Universal Robots URScript: LEscript_grind.script

# File: LEscript_grind.script
# Project: LEonard
# Author: Ned Lecky, Lecky Engineering LLC
# Purpose: LEonard Grinding Support

global version_grind = "LEscript_grind.script 2022-11-23"

global grind_ready = True
# grind_contact_enable:  0=No Contact   1=Touch but no tool/coolant on or force  2=Touch, Tool, Coolant, and Force
global grind_contact_enable = 0
global grind_touch_retract_mm = 3       # How far to retract after touch  (we do 2X this for ghrind_contact_enable=1)
global grind_touch_speed_mmps = 0.1     # How fast to go in for the touch
global grind_force_dwell_ms = 500       # How long to dwell after turning force more on
global grind_max_blend_radius_m = 0.010 # Max blend radius to use while grinding
global grind_trial_speed_mmps = 20      # Grinding speed when not really grinding!
global grind_point_frequency_hz = 4     # Points per second to generate in grind_movel

# Current speeds in use for grinding... the angular are computed off the linear
# And the two are blended by draw_to for cylinders
global grind_linear_vel_mps = 0
global grind_linear_accel_mpss = 0
global grind_linear_blend_radius_m = 0
global grind_angular_vel_rps = 0
global grind_angular_accel_rpss = 0
global grind_angular_blend_radius_rad = 0

# Grinding speeds when not in contact
global grind_jog_speed_mmps = 40     # Speed used internally when adjusting and moving around part
global grind_jog_accel_mmpss = 100   # Accel used internally when adjusting and moving around part

# Force mode parameters
global grind_force_mode_damping = 0.0
global grind_force_mode_gain_scaling = 1.0

# Planning points
global p_operator_init = p[0, 0, 0, 0, 0, 0]    # Where we were when operator issued first grind command
global p_contact_init = p[0, 0, 0, 0, 0, 0]     # Where we first contacted the part
global p_contact_center = p[0, 0, 0, 0, 0, 0]   # Computed where center of pattern would be in contact with part

# Set grind variables chosen by command[2]
# Value after set is always returned to socket
def set_grind_variable():
  global grind_ready = False
  socket_send_bool("grind_ready", grind_ready)

  if command[2] == 1:
    global response = "set grind_contact_enable"
    if command[3] >= 0 and command[3] <= 2:
      global grind_contact_enable = ceil(command[3])
    end
    socket_send_number("grind_contact_enable", grind_contact_enable)
  elif command[2] == 2:
    global response = "set grind_touch_retract_mm"
    if command[3] >= 0:
      global grind_touch_retract_mm = ceil(command[3])
    end
    socket_send_number("grind_touch_retract_mm", grind_touch_retract_mm)
  elif command[2] == 3:
    global response = "set grind_touch_speed_mmps"
    if command[3] >= 0:
      global grind_touch_speed_mmps = ceil(command[3])
    end
    socket_send_number("grind_touch_speed_mmps", grind_touch_speed_mmps)
  elif command[2] == 4:
    global response = "set grind_force_dwell_ms"
    if command[3] >= 0:
      global grind_force_dwell_ms = ceil(command[3])
    end
    socket_send_number("grind_force_dwell_ms", grind_force_dwell_ms)
  elif command[2] == 5:
    global response = "set grind_max_wait_ms"
    if command[3] >= 0:
      global grind_max_wait_ms = ceil(command[3])
    end
    socket_send_number("grind_max_wait_ms", grind_max_wait_ms)
  elif command[2] == 6:
    global response = "set grind_max_blend_radius_mm"
    if command[3] >= 0:
      global grind_max_blend_radius_m = command[3] / 1000.0
    end
    socket_send_number("grind_max_blend_radius_mm", grind_max_blend_radius_m * 1000.0)
  elif command[2] == 7:
    global response = "set grind_trial_speed_mmps"
    if command[3] > 0:
      global grind_trial_speed_mmps = ceil(command[3])
    end
    socket_send_number("grind_trial_speed_mmps", grind_trial_speed_mmps)
  elif command[2] == 8:
    global response = "set grind_linear_accel_mmpss"
    if command[3] > 0:
      global grind_linear_accel_mpss = ceil(command[3]) / 1000.0
    end
    socket_send_number("grind_linear_accel_mmpss", grind_linear_accel_mpss * 1000.0)
  elif command[2] == 9:
    global response = "set grind_point_frequency_hz"
    if command[3] >= 0:
      global grind_point_frequency_hz = ceil(command[3])
    end
    socket_send_number("grind_point_frequency_hz", grind_point_frequency_hz)
  elif command[2] == 10:
    global response = "set grind_jog_speed_mmps"
    if command[3] >= 0:
      global grind_jog_speed_mmps = ceil(command[3])
    end
    socket_send_number("grind_jog_speed_mmps", grind_jog_speed_mmps)
  elif command[2] == 11:
    global response = "set grind_jog_accel_mmpss"
    if command[3] >= 0:
      global grind_jog_accel_mmpss = ceil(command[3])
    end
    socket_send_number("grind_jog_accel_mmpss", grind_jog_accel_mmpss)
  elif command[2] == 12:
    global response = "set grind_force_mode_damping"
    if command[3] >= 0:
      global grind_force_mode_damping = limiter(command[3], 0.0, 1.0)
    end
    socket_send_number("grind_force_mode_damping", grind_force_mode_damping)
  elif command[2] == 13:
    global response = "set grind_force_mode_gain_scaling"
    if command[3] >= 0:
      global grind_force_mode_gain_scaling = limiter(command[3], 0.0, 2.0)
    end
    socket_send_number("grind_force_mode_gain_scaling", grind_force_mode_gain_scaling)
  else:
    global response = "Unknown grind set variable command"
  end

  global grind_ready = True
  socket_send_bool("grind_ready", grind_ready)
end
global grind_force_mode_damping = 0.0
global grind_force_mode_gain_scaling = 1.0

# Execute the desired grind operation as specified in command[2]...
def grind():
  global grind_ready = False
  socket_send_bool("grind_ready", grind_ready)

  start_listen_halt_thread()

  global grind_cycle = 0
  socket_send_number("grind_cycle", grind_cycle)

  # Install tcp that puts tcp at center of part (noop for flat parts!)
  iset_tcp(robot_tcp_part)

  if command[2] == 10:
    # LINEAR GRIND
    global response = "grind_line"
    global grind_dx_mm = limiter(command[3], -1000, 1000)
    global grind_dy_mm = limiter(command[4], -1000, 1000)
    n_cycle_setter(command[5])
    speed_setter(command[6], 0)
    global grind_force_N = limiter(command[7], 0, 100)
    global grind_continue = command[8] > 0
    imover_realtime(True)
    grind_line(grind_dx_mm, grind_dy_mm, grind_n_cycles, grind_continue)

  elif command[2] == 11:
    # LINEAR ANGLE GRIND
    global response = "grind_line_deg"
    global grind_len_mm = limiter(command[3], 0, 1000)
    global grind_angle_deg = limiter(command[4], 0, 360)
    n_cycle_setter(command[5])
    speed_setter(command[6], 0)
    global grind_force_N = limiter(command[7], 0, 100)
    global grind_continue = command[8] > 0
    imover_realtime(True)
    global grind_dx_mm = grind_len_mm * cos(d2r(grind_angle_deg))
    global grind_dy_mm = grind_len_mm * sin(d2r(grind_angle_deg))
    grind_line(grind_dx_mm, grind_dy_mm, grind_n_cycles, grind_continue)

  elif command[2] == 20:
    # RECTANGULAR GRIND
    global response = "grind_rect"
    global grind_dx_mm = limiter(command[3], 0, 1000)
    global grind_dy_mm = limiter(command[4], 0, 1000)
    n_cycle_setter(command[5])
    speed_setter(command[6], 0)
    global grind_force_N = limiter(command[7], 0, 100)
    global grind_continue = command[8] > 0
    imover_realtime(True)
    grind_rect(grind_dx_mm, grind_dy_mm, grind_n_cycles, grind_continue)

  elif command[2] == 30:
    # SERPENTINE GRIND
    global response = "grind_serpentine"
    global grind_dx_mm = limiter(command[3], 1, 1000)
    global grind_dy_mm = limiter(command[4], 1, 1000)
    global grind_n_xsteps = limiter(command[5], 1, grind_dx_mm)
    global grind_n_ysteps = limiter(command[6], 1, grind_dy_mm)
    n_cycle_setter(command[7])
    speed_setter(command[8], 0)
    global grind_force_N = limiter(command[9], 0, 10)
    global grind_continue = command[10] > 0
    grind_serpentine(grind_dx_mm, grind_dy_mm, grind_n_xsteps, grind_n_ysteps, grind_n_cycles, grind_continue)

  elif command[2] == 40:
    # POLYGON GRIND
    global response = "grind_poly"
    global grind_circle1_diam_mm = limiter(command[3], 0, 1000)
    # Limit number of sides to 2 (line) to diam_mm/10 (100mm circle can have up to 10 sides)
    global grind_n_sides = limiter(command[4], 2, grind_circle1_diam_mm / 10.0)
    n_cycle_setter(command[5])
    speed_setter(command[6], 0)
    global grind_force_N = limiter(command[7], 0, 100)
    global grind_continue = command[8] > 0
    grind_poly(grind_circle1_diam_mm, grind_n_sides, grind_n_cycles, grind_continue)

  elif command[2] == 45:
    # CIRCULAR GRIND
    global response = "grind_circle"
    global grind_circle1_diam_mm = limiter(command[3], 0, 1000)
    n_cycle_setter(command[4])
    local min_feature_mm = max(1, grind_circle1_diam_mm / 5)
    speed_setter(command[5], min_feature_mm, is_circle = True)
    global grind_force_N = limiter(command[6], 0, 100)
    global grind_continue = command[7] > 0
    grind_circle(grind_circle1_diam_mm, grind_n_cycles, grind_continue)

  elif command[2] == 50:
    # SPIRAL GRIND
    global response = "grind_spiral"
    global grind_circle1_diam_mm = limiter(command[3], 2, 1000)
    global grind_circle2_diam_mm = limiter(command[4], 2, 1000)
    global grind_n_revolutions = limiter(command[5], 1, 1000)
    n_cycle_setter(command[6])
    local min_diam_mm = min(grind_circle1_diam_mm, grind_circle2_diam_mm)
    local min_feature_mm = max(1, min_diam_mm / 5)
    speed_setter(command[7], min_feature_mm, is_circle = True)
    global grind_force_N = limiter(command[8], 0, 100)
    global grind_continue = command[9] > 0
    grind_spiral(grind_circle1_diam_mm, grind_circle2_diam_mm, grind_n_revolutions, grind_n_cycles, grind_continue)

  elif command[2] == 99:
    # RETRACT COMMAND
    global response = "grind_retract"
    imover_realtime(True)
    set_grind_process_state(False)
  else:
    # Illegal grind command
    global response = "Unknown grind command"
  end

  # Restore tool-only tcp
  iset_tcp(robot_tcp)

  stop_listen_halt_thread()

  global grind_ready = True
  socket_send_bool("grind_ready", grind_ready)
end

# Set global grind_n_cycles based on whether we really going to grind
def n_cycle_setter(n_cycles):
  if grind_contact_enable == 2:
    global grind_n_cycles = limiter(n_cycles, 0, 100)
  else:
    global grind_n_cycles = limiter(n_cycles, 0, 1)
  end
  socket_send_number("grind_n_cycles", grind_n_cycles)
end

# Set all speed and acceleration globals based on part geometry and whether we really going to grind
def speed_setter(speed_mmps, max_blend_radius_mm = 0.0, is_circle = False):
  speed_mmps = limiter(speed_mmps, 0.1, 400)

  # Figure out best blend radius to use
  # Line, Rect, Serp, and Poly all use r=0 otherwise blend radius causes path sanity failures
  local max_blend_radius_m = max_blend_radius_mm / 1000.0
  global grind_linear_blend_radius_m = min(grind_max_blend_radius_m, max_blend_radius_m)
  if is_circle:
    #if grind_linear_blend_radius_m < 0.001:
    #  grind_linear_blend_radius_m = 0.001
    #end
    grind_linear_blend_radius_m = 0.001
  end

  if grind_contact_enable == 2:
    global grind_linear_vel_mps = speed_mmps / 1000.0
  else:
    global grind_linear_vel_mps = grind_trial_speed_mmps / 1000.0
  end

  # If part is cylinder or spherical, diameter will be >0
  # Set appropriate angular values... even flats need to now how fast to
  # rotate on jog commands!
  local diam_m = robot_part_geometry[1] / 1000.0
  local diam_m = limiter(diam_m, 0.075, 3.0)
  # These are 1/4 the theoretical rotational speeds but we need to set them like this to get the correct speed- why??????
  # rot_vel (rad/s) = linear_vel (m/s) * 2pi (rad/s) / pi * diam (m/s)
  local coeff = 0.5 # Should be 2 and why 0.5 is inexplicable
  global grind_angular_vel_rps = grind_linear_vel_mps * coeff / diam_m
  global grind_angular_accel_rpss = grind_linear_accel_mpss * coeff / diam_m
  global grind_angular_blend_radius_rad = grind_linear_blend_radius_m * coeff / diam_m

  socket_send_number("grind_linear_vel_mmps", grind_linear_vel_mps * 1000.0)
  socket_send_number("grind_linear_accel_mmpss", grind_linear_accel_mpss * 1000.0)
  socket_send_number("grind_linear_blend_radius_mm", grind_linear_blend_radius_m * 1000.0)
  socket_send_number("grind_angular_vel_rps", grind_angular_vel_rps)
  socket_send_number("grind_angular_accel_rpss", grind_angular_accel_rpss)
  socket_send_number("grind_angular_blend_radius_rad", grind_angular_blend_radius_rad)
end

global grind_circle_n_sides = 0
# How many points should we use for a circle diam_m at speed_mps?
def recommend_npoints(diam_m, speed_mps):

  # Calc 1: Interrupt rate
  # Want at least so many points per second
  local circum_m = MATH_PI * diam_m
  local t_circle = circum_m / speed_mps
  global grind_circle_n_sides1 = ceil(t_circle * grind_point_frequency_hz)

  # Calc 2: Smoothness
  # 5mm diam needs 10 pts... so 2X?
  # 100mm diam gets 200 points
  # 1mm diam gets 2 points
  global grind_circle_n_sides2 = ceil(diam_m * 1000 * 2)

  global grind_circle_n_sides3 = 0
  if grind_linear_blend_radius_m > 0.0001:
    # Calc 3: Stay ahead of blend radius
    # Do a point every 2 blend radii
    global grind_circle_n_sides3 = ceil(circum_m / (grind_linear_blend_radius_m * 2))
  end

  # Choose the max and then limit it
  #global grind_circle_n_sides = max(grind_circle_n_sides1, grind_circle_n_sides2)
  #global grind_circle_n_sides = max(grind_circle_n_sides, grind_circle_n_sides3)
  #global grind_circle_n_sides = limiter(grind_circle_n_sides, 2, 2000)

  global grind_circle_n_sides = limiter(grind_circle_n_sides2, 2, 2000)

  return grind_circle_n_sides
end

# Get into contact with part (or away from it)
# enable:  0=No Contact   1=Touch but no tool/coolant on or force  2=Touch, Tool, Coolant, and Force
def contact_part(on = False, enable = 0):
  if on:
    if enable == 0:
      # Just do a small forward motion in the direction of touchoff- this is a simulated p_contact_init
      draw_speed_once(grind_jog_speed_mmps, grind_jog_accel_mmpss)
      p_contact_init = draw_relative(p[0, 0, 0.005, 0, 0, 0])
    elif enable == 1:
      if grind_force_N > 0:
        # Advance until contact but retract 2X grind distance and use this as a simulated p_contact_init
        local success = itouchoff(grind_touch_speed_mmps, grind_touch_retract_mm * 2.0)
        global p_contact_init = iget_actual_tcp_pose()
      else:
        # No Touchoff: p_contact_init is just assumed to be where you are!
        global p_contact_init = iget_actual_tcp_pose()
        local success = True
      end
      return success
    elif enable == 2:
      if grind_force_N > 0:
        # Advance until contact
        local success = itouchoff(grind_touch_speed_mmps, grind_touch_retract_mm)
        # Touchoff has backed off by grind_touch_retract_mm so we need to compute that actual p_contact_init
        global p_contact_init = pose_trans(iget_actual_tcp_pose(), p[0, 0, grind_touch_retract_mm / 1000.0, 0, 0, 0])
      else:
        # No Touchoff: p_contact_init is just assumed to be right in front of you!
        global p_contact_init = pose_trans(iget_actual_tcp_pose(), p[0, 0, grind_touch_retract_mm / 1000.0, 0, 0, 0])
        local success = True
      end
      return success
    end
  else:  # Back away
    # Construct a move back in Z only from here
    draw_speed_once(grind_jog_speed_mmps, grind_jog_accel_mmpss)
    draw_relative(p[0, 0, -0.010, 0, 0, 0])
  end

  return True
end

# Sets digital outpus based 8-element list of 4 pairs DOUT#,State.  -1 indicates unused slot
def set_digital_output_list(list):
  i = 0
  while i < 8:
    if list[i] >= 0:
      b = list[i + 1] == 1
      set_digital_out(list[i], b)
    end
    i = i + 2
  end
end

# Turn tool power on/off if enable=2
def tool_power(on = False, enable = 0):
  if enable < 2:
    return None
  end

  if on:
    # ON IO
    set_digital_output_list(robot_tool_on_outputs)
  else:
    # OFF IO
    set_digital_output_list(robot_tool_off_outputs)
  end

  return None
end

# Turn coolant on/off if enable=2
def coolant_flow(on = False, enable = 0):
  if enable < 2:
    return None
  end

  if on:
    # ON IO
    set_digital_output_list(robot_coolant_on_outputs)
  else:
    # OFF IO
    set_digital_output_list(robot_coolant_off_outputs)
  end

  return None
end

# Turn force mode on/off if enable=2
def apply_force(on = False, enable = 0, force_n = 5, approach_speed_mmps = 10):
  if enable < 2:
    return None
  end

  if on:
    izero_ftsensor()
    if force_n > 0:
      # Standard force mode
      iforce_mode(force_n, approach_speed_mmps)
      sleep(grind_force_dwell_ms / 1000.0)
    else:
      # Move straight to previously estimated p_contact_init (grind_retract_mm ahead of you)
      draw_speed_once(grind_touch_speed_mmps, grind_jog_accel_mmpss)
      draw_relative(p[0, 0, 0, 0, 0, 0])
      global imover_force_N = 0
    end
  else:
    iend_force_mode()
    sleep(0.1)
  end

  return None
end

# Start/Stop Grinding
# Pose to center is the offset we should move to initial touch point [0]=FLAT [1]=CYLINDER [2]=SPHERE
global grind_process_state = False
def set_grind_process_state(on = False, coord_to_center = p[0, 0, 0, 0, 0, 0]):
  set_ok_to_proceed(True)
  if on and not grind_process_state:
    # Need to start the grind
    global p_operator_init = iget_target_tcp_pose()

    izero_ftsensor()

    # TODO This calc isn't exactly right... we will undermove slightly on curved surfaces
    # Think about it
    draw_origin(p_operator_init)
    draw_speed_once(grind_jog_speed_mmps, grind_jog_accel_mmpss)
    drawgi_finish(coord_to_center)
    if not ok_to_proceed():
      set_ok_to_proceed(True)
      draw_speed_once(grind_jog_speed_mmps, grind_jog_accel_mmpss)
      draw_finish(p[0, 0, 0, 0, 0, 0])
      return False
    end

    # Touch part and refine p_contact_init
    local contact_success = contact_part(True, grind_contact_enable)
    if not contact_success:
      # Never hit the part (searches 25mm down)
      set_ok_to_proceed(True)
      draw_speed_once(grind_jog_speed_mmps, grind_jog_accel_mmpss)
      draw_finish(p[0, 0, 0, 0, 0, 0])
      return False
    end

    # Compute p_contact_center... where we would have been if we had touched off from the operator teach position!
    local  reverse_coord_to_center = coord_to_center
    local i = 0
    while i < 6:
      reverse_coord_to_center[i] = -reverse_coord_to_center[i]
      i = i + 1
    end
    global p_contact_center = pose_trans(p_contact_init, draw_geometry_compensate(reverse_coord_to_center))

    # All remaining grind moves will be relative to this computed center point
    draw_origin(p_contact_center)

    # Now power everything on (although these will do nothing unless contact_enable==2)
    tool_power(True, grind_contact_enable)
    coolant_flow(True, grind_contact_enable)
    drawgi_finish(coord_to_center)
    apply_force(True, grind_contact_enable, grind_force_N, grind_touch_speed_mmps)

    if not ok_to_proceed():
      terminate_grind()
      return False
    end

    global grind_process_state = True
    socket_send_bool("grind_process_state", grind_process_state)
    return True
  elif on and grind_process_state:
    # Continuing a grind...

    # Move to initial grind position relative to initial p_contact_center
    # Stay at current speeds
    drawgi_finish(coord_to_center)
    if not ok_to_proceed():
      terminate_grind()
      return False
    end

    # Need to change force?
    # Lift, rezero, and then head toward start of next pattern
    if grind_contact_enable == 2 and imover_force_N != grind_force_N:
      # This would be great, but the sensor drifts and forces returned by get_tcp_force() are offset
      #iforce_update(grind_force_N, grind_touch_speed_mmps)

      # So we do a full reset!
      iend_force_mode()
      draw_speed_once(grind_jog_speed_mmps, grind_jog_accel_mmpss)
      draw_relative(p[0, 0, -0.004, 0, 0, 0])
      if not ok_to_proceed():
        terminate_grind()
        return False
      end
      sleep(1)
      if not ok_to_proceed():
        terminate_grind()
        return False
      end

      if grind_force_N > 0:
        # Switching to force>0
        izero_ftsensor()
        iforce_mode(grind_force_N, grind_touch_speed_mmps)
        sleep(grind_force_dwell_ms / 1000.0)
      else:
        # Switching to force=0
        draw_speed_once(grind_jog_speed_mmps, grind_jog_accel_mmpss)
        draw_relative(p[0, 0, 0.004, 0, 0, 0])
      end
    end
    return True
  elif not on and grind_process_state:
    terminate_grind()
    return True
  end

  # If you fall through, send state update!
  socket_send_bool("grind_process_state", grind_process_state)
  return False
end

def terminate_grind():
  set_ok_to_proceed(True)
  #imover_realtime(True)

  # Shut everything down and return to original pose
  apply_force(False, grind_contact_enable, 0)
  contact_part(False, grind_contact_enable)
  coolant_flow(False, grind_contact_enable)
  tool_power(False, grind_contact_enable)

  # Always end with a move back to origin
  draw_speed_once(grind_jog_speed_mmps, grind_jog_accel_mmpss)
  draw_origin(p_operator_init)
  draw_sync_current_dp(iget_actual_tcp_pose())
  draw_finish(p[0, 0, 0, 0, 0, 0])

  global grind_process_state = False
  socket_send_bool("grind_process_state", grind_process_state)
end

######################################################################################
# START TOP LEVEL GRIND FUNCTIONS AND THEIR PATTERNS
#
# Grind along a line dx_mm x dy_mm centered on current tool position. Repeat n_cycles times. If stay_in_contact, stay_in_contact at end.
def grind_line(dx_mm, dy_mm, n_cycles, stay_in_contact):
  if n_cycles < 1:
    return True
  end

  local dx_m = dx_mm / 1000.0
  local dy_m = dy_mm / 1000.0

  # Grind time estimate
  local time_ms = sqrt(dx_mm * dx_mm + dy_mm * dy_mm) * n_cycles / grind_linear_vel_mps + 1500
  socket_send_number("robot_step_time_estimate_ms", time_ms)

  imover_realtime(True)
  if not set_grind_process_state(True, pattern_line(dx_m, dy_m, n_cycles, True)):
    return False
  end

  # Grind the pattern
  start_user_timer()
  pattern_line(dx_m, dy_m, n_cycles)
  stop_user_timer()

  if not stay_in_contact or not ok_to_proceed():
    set_grind_process_state(False)
  end

  return True
end

# Move along a line dx_m x dy_m. Repeat n_cycles times.
# If return_initial_offset_only, just returns dp to initial drawing point
# Move in x direction first, then y
def pattern_line(dx_m, dy_m, n_cycles, return_initial_offset_only = False):
  local x2 = dx_m / 2.0
  local y2 = dy_m / 2.0

  global dp1 = p[-x2, -y2, 0, 0, 0, 0]
  global dp2 = p[x2, y2, 0, 0, 0, 0]

  if return_initial_offset_only:
    return dp1
  end


  # Cyline calibration is all done using lines on cylinders
  local shape = robot_part_geometry[0]
  local is_cylinder = shape == 2
  if is_cylinder and cyline_cal_enabled:
    start_cal_timer()
  end

  global grind_cycle = 1
  local dpdest = dp2
  while (ok_to_proceed() and grind_cycle <= n_cycles):
    socket_send_number("grind_cycle", grind_cycle)

    drawgi_finish(dpdest)

    if dpdest == dp1:
      dpdest = dp2
    else:
      dpdest = dp1
    end

    grind_cycle = grind_cycle + 1
  end

  # Cyline calibration cleanup
  if is_cylinder and cyline_cal_enabled:
    local t = stop_cal_timer()
    adjust_cyline_coefficient(t)
  end

  return dp1
end


# Grind along a rect dx_mm x dy_mm centered on current tool position. Repeat n_cycles times. If stay_in_contact, stay_in_contact at end.
# Move in x direction first, then y
def grind_rect(dx_mm, dy_mm, n_cycles, stay_in_contact):
  if n_cycles < 1:
    return True
  end

  dx_m = dx_mm / 1000.0
  dy_m = dy_mm / 1000.0
  diam_m = robot_part_geometry[1] / 1000.0
  radius_m = diam_m / 2.0
  drx_rad = dx_m / radius_m
  dry_rad = dy_m / radius_m

  # Grind time estimate
  time_ms = 2 * (dx_mm + dy_mm) * n_cycles / grind_linear_vel_mps + 1500
  socket_send_number("robot_step_time_estimate_ms", time_ms)

  imover_realtime(True)
  if not set_grind_process_state(True, pattern_rect(dx_m, dy_m, n_cycles, True)):
    return False
  end

  # Grind the pattern
  start_user_timer()
  pattern_rect(dx_m, dy_m, n_cycles)
  stop_user_timer()

  if not stay_in_contact or not ok_to_proceed():
    set_grind_process_state(False)
  end

  return True
end

# Move along a rect dx_m x dy_m. Repeat n_cycles times.
# If return_initial_offset_only, just returns dp to initial drawing point
# Move in x direction first, then y
def pattern_rect(dx_m, dy_m, n_cycles, return_initial_offset_only = False):
  local x2 = dx_m / 2.0
  local y2 = dy_m / 2.0

  # Compute chamfer size. Use max_blend_radius unless it is < 1/3 the smallest dim
  # Example: On 20mm rects, 2mm chamfer is as large as looks reasonable
  local dx = grind_max_blend_radius_m
  local dx = min(dx, dx_m / 10)
  local dx = min(dx, dy_m / 10)

  global dp1 = p[-x2, -y2, 0, 0, 0, 0]
  global dp1a = dp1
  global dp1b = dp1
  dp1a[1] = dp1a[1] + dx
  dp1b[0] = dp1b[0] + dx

  global dp2 = p[x2, -y2, 0, 0, 0, 0]
  global dp2a = dp2
  global dp2b = dp2
  dp2a[0] = dp2a[0] - dx
  dp2b[1] = dp2b[1] + dx

  global dp3 = p[x2, y2, 0, 0, 0, 0]
  global dp3a = dp3
  global dp3b = dp3
  dp3a[1] = dp3a[1] - dx
  dp3b[0] = dp3b[0] - dx

  global dp4 = p[-x2, y2, 0, 0, 0, 0]
  global dp4a = dp4
  global dp4b = dp4
  dp4a[0] = dp4a[0] + dx
  dp4b[1] = dp4b[1] - dx

  if return_initial_offset_only:
    return dp1b
  end

  global grind_cycle = 1
  while (ok_to_proceed() and grind_cycle <= n_cycles):
    socket_send_number("grind_cycle", grind_cycle)

    # 4-point version (With blend)
    # Fails for blend radius/sanity check when in contact
    #draw_to(dp2)
    #draw_to(dp3)
    #draw_to(dp4)
    #if grind_cycle == n_cycles:
    #  draw_finish(dp1)
    #else:
    #  draw_to(dp1)
    #end

    # 4-point version (Without blend)
    #draw_finish(dp2)
    #draw_finish(dp3)
    #draw_finish(dp4)
    #draw_finish(dp1)

    # 8-point version (With blend)
    # Fails for blend radius/sanity check when in contact
    #draw_to(dp2a)
    #draw_to(dp2b)
    #draw_to(dp3a)
    #draw_to(dp3b)
    #draw_to(dp4a)
    #draw_to(dp4b)
    #draw_to(dp1a)
    #if grind_cycle == n_cycles:
    #  draw_finish(dp1b)
    #else:
    #  draw_to(dp1b)
    #end

    # 8-point version (Without blend)
    drawgi_finish(dp2a)
    drawgi_finish(dp2b)
    drawgi_finish(dp3a)
    drawgi_finish(dp3b)
    drawgi_finish(dp4a)
    drawgi_finish(dp4b)
    drawgi_finish(dp1a)
    drawgi_finish(dp1b)

    grind_cycle = grind_cycle + 1
  end

  return dp1b
end

# Grind along a rect in serpentine dx_mm,dy_mm incrementing by xstep_mm,ystep_mm centered on current tool position. Repeat n_cycles times. If stay_in_contact, stay_in_contact at end.
# Move in x direction first, then y
def grind_serpentine(dx_mm, dy_mm, n_xsteps, n_ysteps, n_cycles, stay_in_contact):
  if n_cycles < 1:
    return True
  end

  # Either n_xsteps or n_ysteps must be 1. Whichever one is one will be the direction of the first move.
  if n_xsteps != 1 and n_ysteps != 1:
    return False
  end

  local dx_m = dx_mm / 1000.0
  local dy_m = dy_mm / 1000.0
  local part_radius_m = robot_part_geometry[1] / 2000.0
  local drx_rad = dx_m / part_radius_m
  local dry_rad = dy_m / part_radius_m

  # Grind time estimate
  # Per Cycle:
  # 1,3 does 4 passes in x and 1 in y     3,1 does 4 passes in Y and 1 in X
  #   ########################            #  ####  #
  #                          #            #  #  #  #
  #   ########################            #  #  #  #
  #   #                                   #  #  #  #
  #   ########################            #  #  #  #
  #                          #            #  #  #  #
  #   ########################            ####  ####
  if n_xsteps == 1:
    time_ms = (dx_mm * (n_ysteps + 1) + dy_mm) * n_cycles / grind_linear_vel_mps + 1500
  else:
    time_ms = (dx_mm + dy_mm * (n_xsteps + 1)) * n_cycles / grind_linear_vel_mps + 1500
  end
  socket_send_number("robot_step_time_estimate_ms", time_ms)

  imover_realtime(True)
  if not set_grind_process_state(True, pattern_serpentine(dx_m, dy_m, n_xsteps, n_ysteps, n_cycles, True)):
    return False
  end

  # Grind the pattern
  start_user_timer()
  pattern_serpentine(dx_m, dy_m, n_xsteps, n_ysteps, n_cycles)
  stop_user_timer()

  if not stay_in_contact or not ok_to_proceed():
    set_grind_process_state(False)
  end

  return True
end

# Move along a serpentine dx_m,dy_m in n_xsteps,n_ysteps. Repeat n_cycles times.
# If return_initial_offset_only, just returns dp to initial drawing point
# Move in direction of whichever nsteps is 1 first
def pattern_serpentine(dx_m, dy_m, n_xsteps, n_ysteps, n_cycles, return_initial_offset_only = False):
  local t_move_x = dx_m / grind_linear_vel_mps
  local t_move_y = dy_m / grind_linear_vel_mps

  # Bottom left corner, grid 0,0
  local x2 = dx_m / 2.0
  local y2 = dy_m / 2.0
  local dp1 = p[-x2, -y2, 0, 0, 0, 0]
  local dp2 = dp1

  if return_initial_offset_only:
    return dp1
  end


  # Track our grid square number... we're in [0,0] and moving [+1,+1] in either x or y
  local x_grid = 0
  local y_grid = 0
  local x_incr = 1
  local y_incr = 1
  local grid_dx_m = dx_m / n_xsteps
  local grid_dy_m = dy_m / n_ysteps

  # How many moves does it take to complete a pass?
  local n_moves_per_pass = (n_xsteps + n_ysteps) * 2 - 1

  local move_count = 0
  global grind_cycle = 1
  while (ok_to_proceed() and grind_cycle <= n_cycles):
    # This will repeat for each leg of the serpentine!
    socket_send_number("grind_cycle", grind_cycle)

    # Skip first X move if we should start with a y move
    if move_count != 0 or n_xsteps == 1:
      # Advance x_grid by x_incr
      x_grid = x_grid + x_incr

      # Move to the corresponding position
      local dc = [x_grid * grid_dx_m - x2, y_grid * grid_dy_m - y2, 0,0,0,0]
      if move_count == n_moves_per_pass:
        drawgi_finish(dc)
      else:
        #draw_to(dp)  # With blend- fails for path sanity/blend failure error when in contact
        drawgi_finish(dc)
      end

      # Adjust x direction
      if x_grid >= n_xsteps:
        x_incr = -1
      elif x_grid <= 0:
        x_incr = 1
      end
      move_count = move_count + 1
    end

    if ok_to_proceed() and move_count < n_moves_per_pass:
      # Advance y_grid by y_incr
      y_grid = y_grid + y_incr

      # Move to the corresponding position
      local dc = [x_grid * grid_dx_m - x2, y_grid * grid_dy_m - y2, 0,0,0,0]
      if move_count == n_moves_per_pass:
        drawgi_finish(dc)
      else:
        #draw_to(dp)  # With blend- fails for path sanity/blend failure error when in contact
        drawgi_finish(dc)
      end

      # Adjust y direction
      if y_grid >= n_ysteps:
        y_incr = -1
      elif y_grid <= 0:
        y_incr = 1
      end
      move_count = move_count + 1
    end

    # Detect when we've covered all the grid squares!
    if move_count >= n_moves_per_pass:
      grind_cycle = grind_cycle + 1
      move_count = 0
    end
  end

  return dp1
end

# Grind along a polygon with circle_diam_mm and n_sides. Repeat n_cycles times. If stay_in_contact, stay_in_contact at end.
def grind_poly(circle_diam_mm, n_sides, n_cycles, stay_in_contact):
  if n_cycles < 1:
    return True
  end

  local circle_diam_m = circle_diam_mm / 1000.0
  local part_diam_m = robot_part_geometry[1] / 1000.0

  # Grind time estimate
  local time_ms = MATH_PI * circle_diam_mm * n_cycles / grind_linear_vel_mps + 1500
  socket_send_number("robot_step_time_estimate_ms", time_ms)

  imover_realtime(True)
  if not set_grind_process_state(True, pattern_poly(circle_diam_m, n_sides, n_cycles, True)):
    return False
  end

  # Grind the pattern
  start_user_timer()
  pattern_poly(circle_diam_m, n_sides, n_cycles)
  stop_user_timer()

  if not stay_in_contact or not ok_to_proceed():
    set_grind_process_state(False)
  end
  return True
end

# Grind along a polygon with circle_diam_m and n_sides. Repeat n_cycles times.
# If return_initial_offset_only, just returns dp to initial drawing point
def pattern_poly(circle_diam_m, n_sides, n_cycles, return_initial_offset_only = False):
  local circle_radius_m = circle_diam_m / 2.0

  local dp1 = p[-circle_diam_m / 2, 0, 0, 0, 0, 0]
  if return_initial_offset_only:
    return dp1
  end

  global grind_cycle = 1
  while (ok_to_proceed() and grind_cycle <= n_cycles):
    socket_send_number("grind_cycle", grind_cycle)
    local i = 0
    while ok_to_proceed() and i <= n_sides:
      local theta = d2r(180.0 + 360.0 * i / n_sides)
      local x = circle_radius_m * cos(theta)
      local y = circle_radius_m * sin(theta)

      local dc = [x, y, 0,0,0,0]
      if not ok_to_proceed() or i == n_sides:
        drawgi_finish(dc)
      else:
        #drawgi_to(dp)  # With blend- fails for path sanity/blend failure error when in contact
        drawgi_finish(dc)
      end
      i = i + 1
    end

    grind_cycle = grind_cycle + 1
  end

  return dp1
end

# Grind along a circle with circle_diam_mm. Repeat n_cycles times. If stay_in_contact, stay_in_contact at end.
def grind_circle(circle_diam_mm, n_cycles, stay_in_contact):
  if n_cycles < 1:
    return True
  end

  local circle_diam_m = circle_diam_mm / 1000.0
  local part_diam_m = robot_part_geometry[1] / 1000.0

  # Grind time estimate
  local time_ms = MATH_PI * circle_diam_mm * n_cycles / grind_linear_vel_mps + 1500
  socket_send_number("robot_step_time_estimate_ms", time_ms)

  imover_realtime(False) # True seems to workl!?
  if not set_grind_process_state(True, pattern_circle(circle_diam_m, n_cycles, True)):
    return False
  end

  # Grind the pattern
  start_user_timer()
  pattern_circle(circle_diam_m, n_cycles)
  stop_user_timer()

  if not stay_in_contact or not ok_to_proceed():
    set_grind_process_state(False)
  end
  return True

  if grind_linear_blend_radius_m > 0.0:
    # Try setting n_sides to 1.5 blend radii
    local circum_m = MATH_PI * circle_diam_mm / 1000.
    global grind_circle_n_sides = ceil(circum_m / (grind_linear_blend_radius_m * 1.5))
  end

  return grind_poly(circle_diam_mm, grind_circle_n_sides, n_cycles, stay_in_contact)
end

# Grind along a circle with circle_diam_m. Repeat n_cycles times.
# If return_initial_offset_only, just returns dp to initial drawing point
def pattern_circle(circle_diam_m, n_cycles, return_initial_offset_only = False):
  local circle_radius_m = circle_diam_m / 2.0
  local n_points = recommend_npoints(circle_diam_m, grind_linear_vel_mps)

  local dp1 = p[-circle_radius_m, 0, 0, 0, 0, 0]
  if return_initial_offset_only:
    return dp1
  end

  global grind_cycle = 1
  while (ok_to_proceed() and grind_cycle <= n_cycles):
    socket_send_number("grind_cycle", grind_cycle)
    local i = 0
    while ok_to_proceed() and i <= n_points:
      local theta = d2r(180.0 + 360.0 * i / n_points)
      local x = circle_radius_m * cos(theta)
      local y = circle_radius_m * sin(theta)

      local dc = [x, y, 0,0,0,0]
      if not ok_to_proceed() or i == n_points:
        drawgi_finish(dc)
      else:
        drawgi_to(dc)
      end
      i = i + 1
    end

    grind_cycle = grind_cycle + 1
  end

  return dp1
end

# Grind along a spiral circle1_diam_mm to circle2_diam_mm in n_revolutions with rotations centered on current tool position. Repeat n_cycles times. If stay_in_contact, stay_in_contact at end.
def grind_spiral(circle1_diam_mm, circle2_diam_mm, n_revolutions, n_cycles, stay_in_contact):
  if n_cycles < 1:
    return True
  end

  local circle1_diam_m = circle1_diam_mm / 1000.0
  local circle2_diam_m = circle2_diam_mm / 1000.0
  local part_diam_m = robot_part_geometry[1] / 1000.0

  # Grind time estimate based on average diam
  local avg_diam_mm = (circle1_diam_mm + circle2_diam_mm) / 2.0
  local time_ms = MATH_PI * avg_diam_mm * n_revolutions * n_cycles / grind_linear_vel_mps + 1500
  socket_send_number("robot_step_time_estimate_ms", time_ms)

  imover_realtime(False) # True fails!?
  if not set_grind_process_state(True, pattern_spiral(circle1_diam_m, circle2_diam_m, n_revolutions, n_cycles, True)):
    return False
  end

  # Grind the pattern
  start_user_timer()
  pattern_spiral(circle1_diam_m, circle2_diam_m, n_revolutions, n_cycles)
  stop_user_timer()

  if not stay_in_contact or not ok_to_proceed():
    set_grind_process_state(False)
  end

  return True
end

# Grind a spiral from diam1 to diam2 in n_revolutions revolutions. Repeat n_cycles times.
# If return_initial_offset_only, just returns dp to initial drawing point
def pattern_spiral(circle1_diam_m, circle2_diam_m, n_revolutions, n_cycles, return_initial_offset_only = False):
  local max_diam_m = max(circle1_diam_m, circle2_diam_m)
  local circle1_radius_m = circle1_diam_m / 2.0
  local circle2_radius_m = circle2_diam_m / 2.0

  local dp1 = p[-circle1_radius_m, 0, 0, 0, 0, 0]
  if return_initial_offset_only:
    return dp1
  end

  global grind_cycle = 1
  while (ok_to_proceed() and grind_cycle <= n_cycles):
    socket_send_number("grind_cycle", grind_cycle)

    # Initial conditions
    local theta = d2r(180.0)
    local r_m = circle1_radius_m
    local revs_completed = 0.0
    local rev_slope = (circle2_radius_m - circle1_radius_m) / n_revolutions
    local move_m = grind_linear_blend_radius_m * 2

    while ok_to_proceed() and revs_completed < n_revolutions:
      local delta_theta = move_m / r_m
      local theta = theta + delta_theta
      local x = r_m * cos(theta)
      local y = r_m * sin(theta)

      local dc = [x, y, 0,0,0,0]
      if not ok_to_proceed() or revs_completed >= n_revolutions:
        drawgi_finish(dc)
      else:
        drawgi_to(dc)
      end

      local revs_completed = revs_completed + delta_theta / (2 * MATH_PI)
      local r_m = circle1_radius_m + rev_slope * revs_completed
    end

    grind_cycle = grind_cycle + 1

    # Next cycle- swap diameters so we go in/out/in etc.
    local old_circle1_radius_m = circle1_radius_m
    local circle1_radius_m = circle2_radius_m
    local circle2_radius_m = old_circle1_radius_m
  end

  return dp1
end
#
# END TOP LEVEL GRIND FUNCTIONS AND THEIR PATTERNS
######################################################################################
